TYPE
    ST_SaveParaRemote :
    STRUCT
        Command : ST_CommandBasic;
        Status  : ST_StatusBasic;
    END_STRUCT
END_TYPE

(* stored: Version 1.1.0.1, ProductVersion 3.1.4024.13
   DUT ST_SaveParaRemote: Id {fb2e1f73-8733-4acc-9684-b822dcb59df7} *)
